{attribute 'linkalways'} 
{attribute 'no_explicit_call' := 'This FB is a CLASS and must be accessed using methods or properties'}
{attribute 'enable_dynamic_creation'}
FUNCTION_BLOCK FINAL MUL_BYTE EXTENDS Node
VAR
	in1 : _BYTE(0);
	in2 : _BYTE(0);
	out : _BYTE(0);
END_VAR

METHOD PUBLIC Clone : I_Node
VAR
	pNode : POINTER TO MUL_BYTE;
END_VAR
pNode := __NEW(MUL_BYTE);
Clone := pNode^;
END_METHOD

METHOD FB_init : BOOL
VAR_INPUT
	bInitRetains : BOOL; // if TRUE, the retain variables are initialized (warm start / cold start)
	bInCopyCode : BOOL;  // if TRUE, the instance afterwards gets moved into the copy code (online change)
END_VAR
AddInput('in1',THIS^.in1);
AddInput('in2',THIS^.in2);
AddOutput('out', THIS^.out);
END_METHOD

METHOD PROTECTED OnExecute
VAR
END_VAR
out.Value := in1.Value * in2.Value;
END_METHOD

END_FUNCTION_BLOCK

(* stored: Version 1.1.0.1, ProductVersion 3.1.4024.15
   POU MUL_BYTE: Id {e6bbc368-fafc-4258-af93-fb5b43c9fa61}, SpecialFunc None
   Folder Constructor: Id {eafc4312-2cd4-435d-b3f4-b4f951be7358}
   Method Clone: Id {4fcf6e14-2b39-4d15-9c2f-2992855a5db9}
   Method FB_init: Id {923e7424-62ec-44aa-9a93-96d2a44ed0ef}
   Method OnExecute: Id {239e94e2-6f6a-4fda-b630-a5184369d069} *)
